FUNCTION_BLOCK DigitalSwitch
VAR_INPUT
	input				: BOOL;
END_VAR
VAR_OUTPUT
	inPos00				: BOOL;
	inPos01				: BOOL;
END_VAR

inPos00 	:= NOT input;
inPos01		:= input;

END_FUNCTION_BLOCK

(* stored: Version 1.1.0.1
   POU DigitalSwitch: Id {7cf7d6ce-542d-42cf-9986-2aae388a3fae}, SpecialFunc None *)
